Universal Robots PolyScope program: AlvarezZavaleta-LuisAlberto-P4_2.urp

Program AlvarezZavaleta-LuisAlberto-P4_2 (installation=default directory=/home/ur/ursim-current/programs/T3 createdIn=5.14.5 lastSavedIn=5.14.5 robotSerialNumber=20195399999)
Calibrated DH parameters: a=[0, -0.24355, -0.2132, 0, 0, 0]; d=[0.15185, 0, 0, 0.13105, 0.08535, 0.0921]; alpha=[1.570796, 0, 0, 1.570796, -1.570796, 0]; deltaTheta=[0, 0, 0, 0, 0, 0]
InitVariablesNode
BeforeStart
  P_ini := get_actual_tcp_pose()
  Alt_ini := 0.05
  Script: P_ini[2] = Alt_ini
  MoveL speed 250 mm/s, acceleration 1200 mm/s^2 (useActiveTCP=true) feature=Base
    Waypoint Variable (Variable): variable=P_ini
  Paso :=  (valueSource=Operator message=Paso mm valueType=Integer)
  Dmin :=  (valueSource=Operator message=Diametro(min) mm valueType=Integer)
  Dmax :=  (valueSource=Operator message=Diametro(max) mm valueType=Integer)
  Ltot :=  (valueSource=Operator message=Longitud(total) mm valueType=Integer)
  Lcon :=  (valueSource=Operator message=Longitud(conica) mm valueType=Integer)
  Wait Sleep waitTime=0.5
Robot Program (runOnlyOnce=true)
  'Pasar el valor a mm'
  Dmin := Dmin/2000
  Dmax := Dmax/2000
  Paso := Paso/4000
  Lcon := Lcon/1000
  Ltot := Ltot/1000
  Lup := Ltot - Lcon
  MidPoint0 := P_ini
  'Usaremos Recorrido para llevar la longitud recorrida'
  Recorrido := 0
  Loop While (checkContinuously=false) expression=Ltot>Recorrido
    If Recorrido<Lcon
      Diametro := Dmin+(Recorrido/Lcon)*(Dmax-Dmin)
    ElseIf Ltot-Lcon≤Recorrido
      Diametro := Dmax-((Recorrido-Lup)/Lcon)*(Dmax-Dmin)
    Else 
      Diametro := Dmax
    distance := p[Diametro,0,Recorrido,0,0,0]
    var_1 := sin(1)
    MidPoint1 := pose_add(MidPoint0,distance )
    Recorrido := Recorrido+Paso
    If Recorrido<Lcon
      Diametro := Dmin+(Recorrido/Lcon)*(Dmax-Dmin)
    ElseIf Ltot-Lcon≤Recorrido
      Diametro := Dmax-((Recorrido-Lup)/Lcon)*(Dmax-Dmin)
    Else 
      Diametro := Dmax
    distance := p[0,Diametro,Recorrido,0,0,0]
    MidPoint2 := pose_add(MidPoint0,distance )
    Recorrido := Recorrido+Paso
    If Recorrido<Lcon
      Diametro := Dmin+(Recorrido/Lcon)*(Dmax-Dmin)
    ElseIf Ltot-Lcon≤Recorrido
      Diametro := Dmax-((Recorrido-Lup)/Lcon)*(Dmax-Dmin)
    Else 
      Diametro := Dmax
    distance := p[-Diametro,0,Recorrido,0,0,0]
    MidPoint3 := pose_add(MidPoint0, distance)
    MoveP speed 250 mm/s, acceleration 1200 mm/s^2 (blendRadius=0.025 useActiveTCP=true) feature=Base
      Waypoint Variable (Variable): variable=MidPoint1
      CircleMove (OrientationMode=UNCONSTRAINED)
        Waypoint Variable (Variable): variable=MidPoint2
        Waypoint Variable (Variable): variable=MidPoint3
    Recorrido := Recorrido+Paso
    If Recorrido<Lcon
      Diametro := Dmin+(Recorrido/Lcon)*(Dmax-Dmin)
    ElseIf Ltot-Lcon≤Recorrido
      Diametro := Dmax-((Recorrido-Lup)/Lcon)*(Dmax-Dmin)
    Else 
      Diametro := Dmax
    distance := p[0,-Diametro,Recorrido,0,0,0]
    MidPoint4 := pose_add(MidPoint0,distance )
    Recorrido := Recorrido+Paso
    If Recorrido<Lcon
      Diametro := Dmin+(Recorrido/Lcon)*(Dmax-Dmin)
    ElseIf Ltot-Lcon≤Recorrido
      Diametro := Dmax-((Recorrido-Lup)/Lcon)*(Dmax-Dmin)
    Else 
      Diametro := Dmax
    distance := p[Diametro,0,Recorrido,0,0,0]
    MidPoint5 := pose_add(MidPoint0,distance )
    MoveP speed 250 mm/s, acceleration 1200 mm/s^2 (blendRadius=0.025 useActiveTCP=true) feature=Base
      Waypoint Variable (Variable): variable=MidPoint3
      CircleMove (OrientationMode=UNCONSTRAINED)
        Waypoint Variable (Variable): variable=MidPoint4
        Waypoint Variable (Variable): variable=MidPoint5
